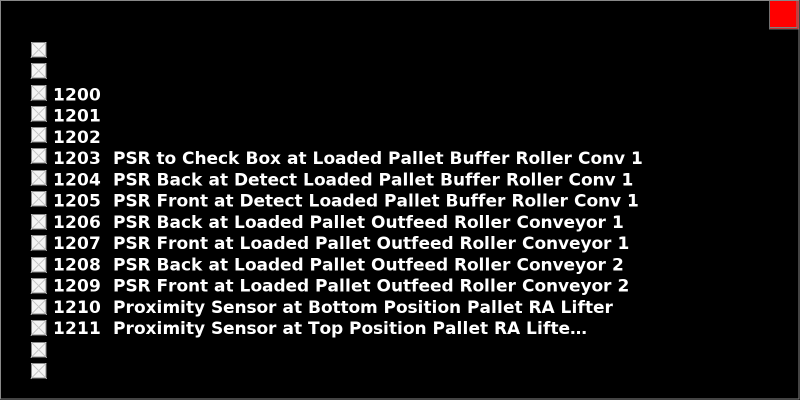
VISUALIZATION P2_DI3  // 800x400, background image 
    ImageSwitcher (31,42 15x15), variable: InputOutput_GVL.Digital_Input[33], behaviour: TOGGLE
    Label (50,16 687x391), "1200 1201 1202 1203 PSR to Check Box at Loaded Pallet Buffer Roller Conv 1 1204 PSR Back at Detect Loaded Pallet Buffer Roller Conv 1 1205 PSR Front at Detect Loaded Pallet Buffer Roller Conv 1 1206 PSR Back at Loaded Pallet Outfeed Roller Conveyor 1 1207 PSR Front at Loaded Pallet Outfeed Roller Conveyor 1 1208 PSR Back at Loaded Pallet Outfeed Roller Conveyor 2 1209 PSR Front at Loaded Pallet Outfeed Roller Conveyor 2 1210 Proximity Sensor at Bottom Position Pallet RA Lifter 1211 Proximity Sensor at Top Position Pallet RA Lifter 1212 PSR Back at Loaded Pallet Outfeed Roller Conveyor 3 1213 PSR Front at Loaded Pallet Outfeed Roller Conveyor 3 1214 PSR Back at Loaded Pallet Outfeed Roller Conveyor 4 1215 PSR Front at Loaded Pallet Outfeed Roller Conveyor 4"
    ImageSwitcher (31,63 15x15), variable: InputOutput_GVL.Digital_Input[34], behaviour: TOGGLE
    ImageSwitcher (31,85 15x15), variable: InputOutput_GVL.Digital_Input[35], behaviour: TOGGLE
    ImageSwitcher (31,106 15x15), variable: InputOutput_GVL.Digital_Input[36], behaviour: TOGGLE
    ImageSwitcher (31,127 15x15), variable: InputOutput_GVL.Digital_Input[37], behaviour: TOGGLE
    ImageSwitcher (31,148 15x15), variable: InputOutput_GVL.Digital_Input[38], behaviour: TOGGLE
    ImageSwitcher (31,170 15x15), variable: InputOutput_GVL.Digital_Input[39], behaviour: TOGGLE
    ImageSwitcher (31,191 15x15), variable: InputOutput_GVL.Digital_Input[40], behaviour: TOGGLE
    ImageSwitcher (31,214 15x15), variable: InputOutput_GVL.Digital_Input[41], behaviour: TOGGLE
    ImageSwitcher (31,235 15x15), variable: InputOutput_GVL.Digital_Input[42], behaviour: TOGGLE
    ImageSwitcher (31,257 15x15), variable: InputOutput_GVL.Digital_Input[43], behaviour: TOGGLE
    ImageSwitcher (31,278 15x15), variable: InputOutput_GVL.Digital_Input[44], behaviour: TOGGLE
    ImageSwitcher (31,299 15x15), variable: InputOutput_GVL.Digital_Input[45], behaviour: TOGGLE
    ImageSwitcher (31,320 15x15), variable: InputOutput_GVL.Digital_Input[46], behaviour: TOGGLE
    ImageSwitcher (31,342 15x15), variable: InputOutput_GVL.Digital_Input[47], behaviour: TOGGLE
    ImageSwitcher (31,363 15x15), variable: InputOutput_GVL.Digital_Input[48], behaviour: TOGGLE
    Button (769,-1 30x30), image: VisuSymbols.Symbols.Wrong
        OnMouseClick: CloseDialog Dialog=P2_DI3, Result=OK, NumpadKeypadSet=True
END_VISUALIZATION

(* stored: Version 1.1.0.1, ProductVersion 3.1.4024.12
   Visu P2_DI3: Id {cbe42f47-a073-4bed-93ec-6d8f2ab859d3} *)
